// TIA Portal V17 export
// export: Created 2024-09-15T12:30:16.6321461Z, ExportSetting WithDefaults, DisplayName Totally Integrated Automation Portal, DisplayVersion V17, DisplayName TIA Portal Openness, DisplayVersion V17, DisplayName TIA Portal Version Control Interface, DisplayVersion V17, DisplayName STEP 7 Professional, DisplayVersion V17, DisplayName STEP 7 Safety, DisplayVersion V17, DisplayName WinCC Professional, DisplayVersion V17
DATA_BLOCK "Copy_Simulation_Variables_DB"   // DB47
VERSION : 0.1
// stored: AutoNumber true, DBAccessibleFromOPCUA true, DBAccessibleFromWebserver true, InstanceOfName Copy_Simulation_Variables, InstanceOfType FB
"Copy_Simulation_Variables"
BEGIN
END_DATA_BLOCK
